(* IEC 61131-3 sources: RL_MAR/experiments/comparison/autoplc/results/gpt-4o-mini_20260511_164212/med_44, 1 file *)

(* ---- med_44_1.st ---- *)
FUNCTION_BLOCK DroneChargingStation
VAR_INPUT
    Drone1BatteryLevel : INT := 0; (* Battery level of Drone 1 (0-100%) *)
    Drone2BatteryLevel : INT := 0; (* Battery level of Drone 2 (0-100%) *)
    Drone3BatteryLevel : INT := 0; (* Battery level of Drone 3 (0-100%) *)
    ChargingTime : TIME := T#30s; (* Charging time required for each drone *)
END_VAR
VAR_OUTPUT
    Drone1Status : BOOL := FALSE; (* Status of Drone 1 *)
    Drone2Status : BOOL := FALSE; (* Status of Drone 2 *)
    Drone3Status : BOOL := FALSE; (* Status of Drone 3 *)
    ChargingStationStatus : BOOL := FALSE; (* Charging station status *)
    DroneDeployed : BOOL := FALSE; (* Indicates if a drone is deployed *)
END_VAR
VAR
    TimeRemaining : TIME := ChargingTime; (* Remaining charging time for the current charging operation *)
    DroneCharging : INT := 0; (* Variable to track which drone is charging: 0 = none, 1 = Drone1, 2 = Drone2, 3 = Drone3 *)
END_VAR

// Initialization
IF NOT ChargingStationStatus THEN
    // Check battery levels and start charging if necessary
    IF Drone1BatteryLevel < 20 AND DroneCharging = 0 THEN
        Drone1Status := TRUE;
        ChargingStationStatus := TRUE;
        TimeRemaining := ChargingTime;
        DroneCharging := 1;
    ELSIF Drone2BatteryLevel < 20 AND DroneCharging = 0 THEN
        Drone2Status := TRUE;
        ChargingStationStatus := TRUE;
        TimeRemaining := ChargingTime;
        DroneCharging := 2;
    ELSIF Drone3BatteryLevel < 20 AND DroneCharging = 0 THEN
        Drone3Status := TRUE;
        ChargingStationStatus := TRUE;
        TimeRemaining := ChargingTime;
        DroneCharging := 3;
    END_IF
END_IF

// Charging Process
IF ChargingStationStatus THEN
    // Decrement the remaining charging time
    TimeRemaining := TimeRemaining - T#1s; // Assuming this block is called every second

    // Check if charging time has elapsed
    IF TimeRemaining <= T#0s THEN
        Drone1Status := FALSE;
        Drone2Status := FALSE;
        Drone3Status := FALSE;
        ChargingStationStatus := FALSE;
        DroneCharging := 0; // Reset charging status
    END_IF
END_IF

// Deployment Monitoring
IF DroneDeployed THEN
    // Check battery levels for deployed drones
    IF Drone1BatteryLevel < 10 THEN
        DroneDeployed := FALSE; // Recall Drone 1
    ELSIF Drone2BatteryLevel < 10 THEN
        DroneDeployed := FALSE; // Recall Drone 2
    ELSIF Drone3BatteryLevel < 10 THEN
        DroneDeployed := FALSE; // Recall Drone 3
    END_IF
END_IF

END_FUNCTION_BLOCK
